	FUNCTION_BLOCK FB 324
	TITLE =G224M COUPLING DEVICE WALL GERM 7
	//COPYRIGHT:    (C) 2009  BUHLER AG, CH-9240 UZWIL, SWITZERLAND
	//
	//PRODUCT:      WinCoS_BIW01_09
	//
	//TITLE:        COUPLING DEVICE WALL GERM 7
	//                Machine group control
	//                Maschinengruppensteuerung
	//
	//--------------------------------------------------------------------------------
	//
	//IDENT:        AUTHOR:             DEPT:                              DATE:
	//
	//P01_FB324.1.0 K.Renz              CSB41                              13.Jan.2010
	//             1st Release
	//
	//--------------------------------------------------------------------------------
	//
	//PURPOSE:
	//
	//MANUAL :
	//
	//RESTRICTIONS:
	//
	//--------------------------------------------------------------------------------
	AUTHOR  : KR
	FAMILY  : USW
	VERSION : 9.9


	VAR
	  Gr       : FB10;	//Standard interface to group
	  InOutValue1    : DINT; //Data for user
	  InOutValue2    : DINT; //Data for user
	  OutWayConflict : BOOL;	//Data for user
	  OutSelectionOk : BOOL;	//Data for user
	  CmdNewValue : BOOL;	//Data for user
	  CmdNewJob   : BOOL;	//Data for user
	  OutCodeOK   : BOOL;	//Data for user
	  InEndOfJob  : BOOL ;	//Data for user
	  staWayOk      : BOOL ;	//Data for user
	  EdgeStartRelease : BOOL ;	//Data for user
	  USW8  : BOOL;	//Data for user
	  USW9 : BOOL;	//Data for user
	  USW10: BOOL;	//Data for user
	  USW11: BOOL;	//Data for user
	  USW12: BOOL;	//Data for user
	  USW13: BOOL;	//Data for user
	  USW14: BOOL;	//Data for user
	  USW15: BOOL;	//Data for user
	     #A_2715_BZS42 : FB14;   // DigInpCont
	     #A_2715_BZS43 : FB14;   // DigInpCont
	     #A_2715_BZS47 : FB14;   // DigInpCont
	     #A_2715_BZS46 : FB14;   // DigInpCont
	     #A_2715_MXZ41 : FB12;   // Motor
	     #A_2715_MXZ45 : FB12;   // Motor
	END_VAR
	VAR_TEMP
	   tmpEnable		: BOOL;
	   tmpFlag  		: BOOL;
	   tmpCmdNext		: BOOL;
	   tmpLocal  		: BOOL;
	   tmpAspOk  		: BOOL;
	   tmpHWStop 		: BOOL;
	   tmpInstanzDBNo       : INT ;
	END_VAR
	BEGIN
	NETWORK
	TITLE =
	NETWORK
	TITLE =Read command from group control
	//Parameter
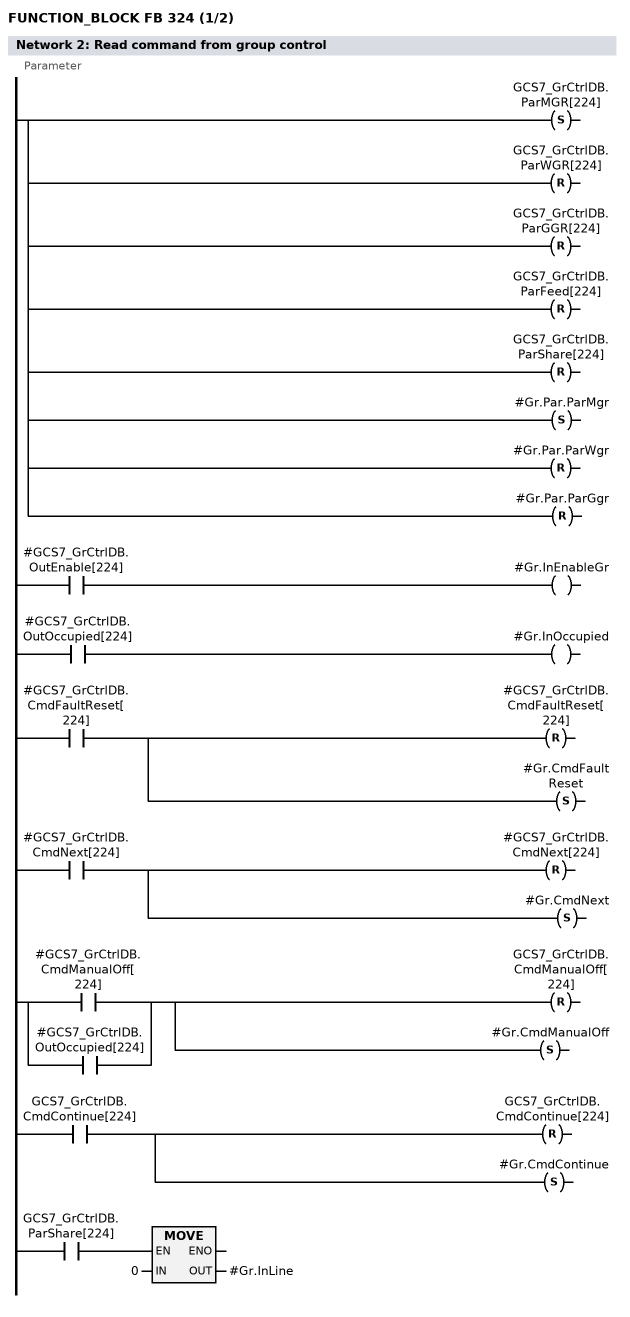
	      SET;
	      S   GCS7_GrCtrlDB.ParMGR[224];
	      R   GCS7_GrCtrlDB.ParWGR[224];
	      R   GCS7_GrCtrlDB.ParGGR[224];
	      R   GCS7_GrCtrlDB.ParFeed[224];
	      R   GCS7_GrCtrlDB.ParShare[224];
	      S   #Gr.Par.ParMgr;
	      R   #Gr.Par.ParWgr;
	      R   #Gr.Par.ParGgr;
	//Command
	      U   #GCS7_GrCtrlDB.OutEnable[224];
	      =   #Gr.InEnableGr;
	      U   #GCS7_GrCtrlDB.OutOccupied[224];
	      =   #Gr.InOccupied;
	      U   #GCS7_GrCtrlDB.CmdFaultReset[224];
	      R   #GCS7_GrCtrlDB.CmdFaultReset[224];
	      S   #Gr.CmdFaultReset;
	      U  #GCS7_GrCtrlDB.CmdNext[224];
	      R   #GCS7_GrCtrlDB.CmdNext[224];
	      S   #Gr.CmdNext;
	      U   #GCS7_GrCtrlDB.CmdManualOff[224];
	      O   #GCS7_GrCtrlDB.OutOccupied[224];
	      R   GCS7_GrCtrlDB.CmdManualOff[224];
	      S   #Gr.CmdManualOff;
	      U  GCS7_GrCtrlDB.CmdContinue[224];
	      R   GCS7_GrCtrlDB.CmdContinue[224];
	      S   #Gr.CmdContinue;
	//Init Line Number
	      U   GCS7_GrCtrlDB.ParShare[224];
	      SPBN WE00;
	      L     0;
	      T     #Gr.InLine;
	WE00: NOP   0;
	NETWORK
	TITLE =Call Methode Control
	// 1. Handle Interface PCControl
	// 2. Prepare mode --> ModePassive,ModeActive,ModeIdling
	// 3. Reset global flags of the group
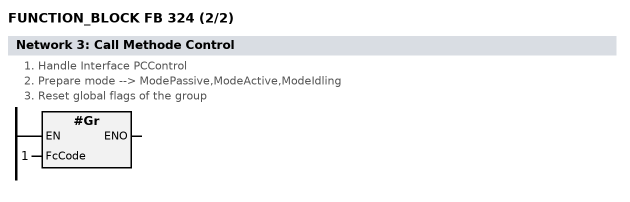
	      CALL #Gr (
	           FcCode                   := 1);
	NETWORK
	TITLE =Restart Idling Time
		L  #Gr.Par.ParIdling;
		L  2;
		>=I;
		SPB IdTm;
		T  #Gr.Par.ParIdling;
	IdTm:   NOP 0;
	      CLR;
	      S    #Gr.CmdRestartIdling;
	NETWORK
	TITLE =Prepare global flags
	NETWORK
	TITLE =Set Pattern (Target position)
	NETWORK
	TITLE =Interlocking WayOk
	//
	NETWORK
	TITLE =Interlocking Autostart
		CLR;
		R   #Gr.OutAutostart;
	NETWORK
	TITLE =Interlocking Enable
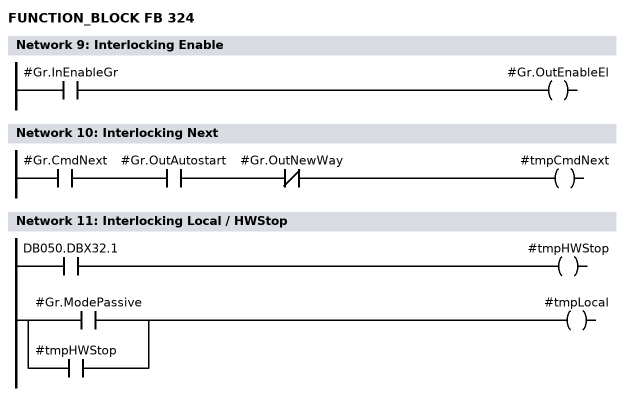
	      U     #Gr.InEnableGr;
	      =     #Gr.OutEnableEl;

	NETWORK
	TITLE =Interlocking Next
	      U     #Gr.CmdNext;
	      U     #Gr.OutAutostart;
	      UN    #Gr.OutNewWay;
	      =    #tmpCmdNext;

	NETWORK
	TITLE =Interlocking Local / HWStop
	      U    DB050.DBX32.1;
	      =    #tmpHWStop;

	      U    #Gr.ModePassive;
	      O    #tmpHWStop;
	      =    #tmpLocal;

	NETWORK
	TITLE ==A-2715-BZS42 : COUPLING DRIVE UNLOCKED
	NOP 0;
	//-InLocal---
	      U     #tmpLocal;
	      =     #A_2715_BZS42.InLocal;
	//
	//-Monitoring---
	      CLR;
	      =      #A_2715_BZS42.InMonTrue;
	      CLR;
	      =      #A_2715_BZS42.InMonFalse;
	//
	//-PreAlarm---
	      CLR;
	      =      #A_2715_BZS42.InPreAlarmTrue;
	      CLR;
	      =      #A_2715_BZS42.InPreAlarmFalse;
	//
	//-Additional commands---
	//      CLR
	//      S     #A_2715_BZS42.CmdRunTimeOutTime
	//
	//-Read inputs---
	      U     E 763.0;
	      =     #A_2715_BZS42.InpTrue;
	      U   DB050.DBX32.1;
	      =     #A_2715_BZS42.InHWStop;
	       U     PLC_DPInfo.Master[1].SlavesError[75];
	       =       #A_2715_BZS42.InDPFault;
	//
	//-Set Parameters---
	//
	//-Call object control---
	      CALL  #A_2715_BZS42;
	//
	//-Write outputs---
	NETWORK
	TITLE ==A-2715-BZS43 : COUPLING DRIVE LOCKED
	NOP 0;
	//-InLocal---
	      U     #tmpLocal;
	      =     #A_2715_BZS43.InLocal;
	//
	//-Monitoring---
	      CLR;
	      =      #A_2715_BZS43.InMonTrue;
	      CLR;
	      =      #A_2715_BZS43.InMonFalse;
	//
	//-PreAlarm---
	      CLR;
	      =      #A_2715_BZS43.InPreAlarmTrue;
	      CLR;
	      =      #A_2715_BZS43.InPreAlarmFalse;
	//
	//-Additional commands---
	//      CLR
	//      S     #A_2715_BZS43.CmdRunTimeOutTime
	//
	//-Read inputs---
	      U     E 763.1;
	      =     #A_2715_BZS43.InpTrue;
	      U   DB050.DBX32.1;
	      =     #A_2715_BZS43.InHWStop;
	       U     PLC_DPInfo.Master[1].SlavesError[75];
	       =       #A_2715_BZS43.InDPFault;
	//
	//-Set Parameters---
	//
	//-Call object control---
	      CALL  #A_2715_BZS43;
	//
	//-Write outputs---
	NETWORK
	TITLE ==A-2715-BZS47 : COUPLING DRIVE LOCKED
	NOP 0;
	//-InLocal---
	      U     #tmpLocal;
	      =     #A_2715_BZS47.InLocal;
	//
	//-Monitoring---
	      CLR;
	      =      #A_2715_BZS47.InMonTrue;
	      CLR;
	      =      #A_2715_BZS47.InMonFalse;
	//
	//-PreAlarm---
	      CLR;
	      =      #A_2715_BZS47.InPreAlarmTrue;
	      CLR;
	      =      #A_2715_BZS47.InPreAlarmFalse;
	//
	//-Additional commands---
	//      CLR
	//      S     #A_2715_BZS47.CmdRunTimeOutTime
	//
	//-Read inputs---
	      U     E 763.3;
	      =     #A_2715_BZS47.InpTrue;
	      U   DB050.DBX32.1;
	      =     #A_2715_BZS47.InHWStop;
	       U     PLC_DPInfo.Master[1].SlavesError[75];
	       =       #A_2715_BZS47.InDPFault;
	//
	//-Set Parameters---
	//
	//-Call object control---
	      CALL  #A_2715_BZS47;
	//
	//-Write outputs---
	NETWORK
	TITLE ==A-2715-BZS46 : COUPLING DRIVE UNLOCKED
	NOP 0;
	//-InLocal---
	      U     #tmpLocal;
	      =     #A_2715_BZS46.InLocal;
	//
	//-Monitoring---
	      CLR;
	      =      #A_2715_BZS46.InMonTrue;
	      CLR;
	      =      #A_2715_BZS46.InMonFalse;
	//
	//-PreAlarm---
	      CLR;
	      =      #A_2715_BZS46.InPreAlarmTrue;
	      CLR;
	      =      #A_2715_BZS46.InPreAlarmFalse;
	//
	//-Additional commands---
	//      CLR
	//      S     #A_2715_BZS46.CmdRunTimeOutTime
	//
	//-Read inputs---
	      U     E 763.2;
	      =     #A_2715_BZS46.InpTrue;
	      U   DB050.DBX32.1;
	      =     #A_2715_BZS46.InHWStop;
	       U     PLC_DPInfo.Master[1].SlavesError[75];
	       =       #A_2715_BZS46.InDPFault;
	//
	//-Set Parameters---
	//
	//-Call object control---
	      CALL  #A_2715_BZS46;
	//
	//-Write outputs---
	NETWORK
	TITLE ==A-2715-MXZ41 : WALL COUPLING DRIVE
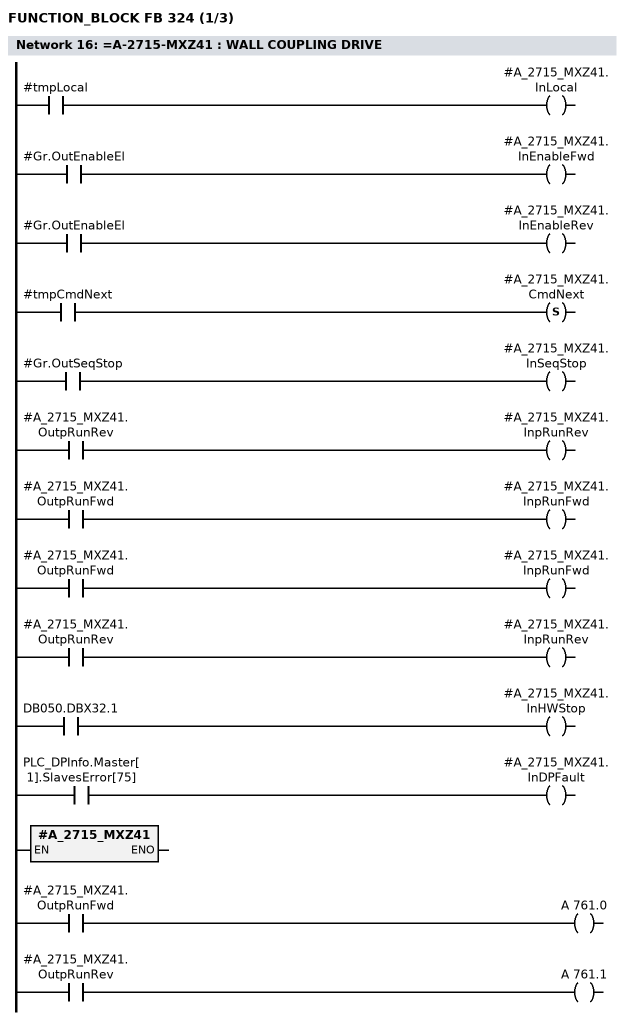
	NOP 0;
	//-InLocal---
	      U     #tmpLocal;
	      =     #A_2715_MXZ41.InLocal;
	//
	//-Interlocking---
	      U     #Gr.OutEnableEl;
	      =     #A_2715_MXZ41.InEnableFwd;
	      U     #Gr.OutEnableEl;
	      =     #A_2715_MXZ41.InEnableRev;
	//
	      U    #tmpCmdNext;
	      S     #A_2715_MXZ41.CmdNext;
	//
	      U     #Gr.OutSeqStop;
	      =     #A_2715_MXZ41.InSeqStop;
	//
	//-Read inputs---
	      U     #A_2715_MXZ41.OutpRunRev;
	      =     #A_2715_MXZ41.InpRunRev;
	      U     #A_2715_MXZ41.OutpRunFwd;
	      =     #A_2715_MXZ41.InpRunFwd;
	      U     #A_2715_MXZ41.OutpRunFwd;
	      =     #A_2715_MXZ41.InpRunFwd;
	      U     #A_2715_MXZ41.OutpRunRev;
	      =     #A_2715_MXZ41.InpRunRev;
	      U   DB050.DBX32.1;
	      =     #A_2715_MXZ41.InHWStop;
	       U     PLC_DPInfo.Master[1].SlavesError[75];
	       =       #A_2715_MXZ41.InDPFault;
	//
	//-Set Parameters---
	//
	//-Call object control---
	      CALL  #A_2715_MXZ41;
	//
	//-Write outputs---
	      U     #A_2715_MXZ41.OutpRunFwd;
	      =     A 761.0;
	      U     #A_2715_MXZ41.OutpRunRev;
	      =     A 761.1;
	NETWORK
	TITLE ==A-2715-MXZ45 : WALL COUPLING DRIVE
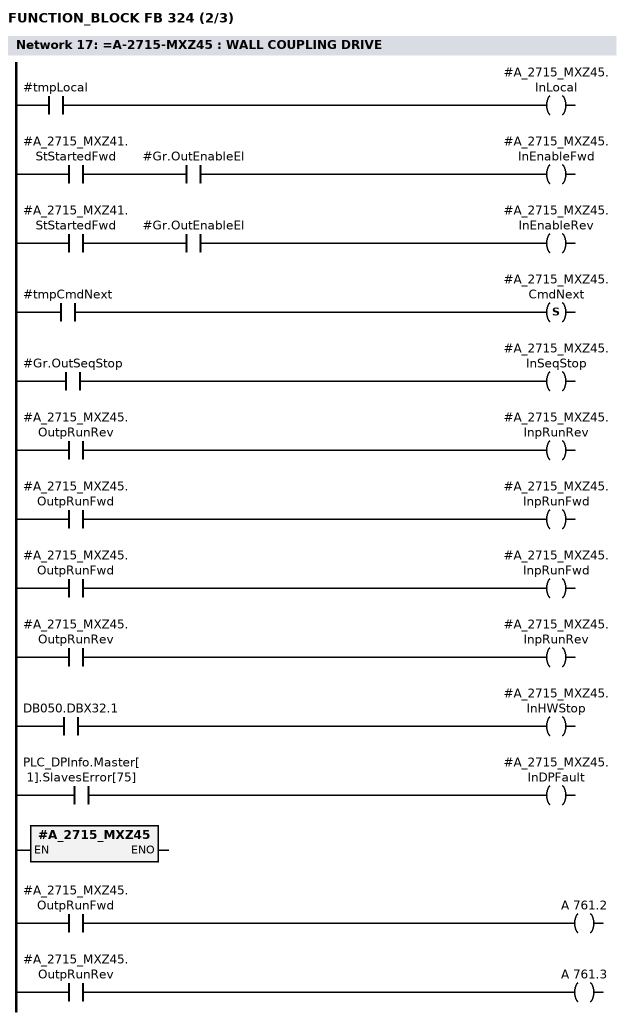
	NOP 0;
	//-InLocal---
	      U     #tmpLocal;
	      =     #A_2715_MXZ45.InLocal;
	//
	//-Interlocking---
	      U     #A_2715_MXZ41.StStartedFwd;
	      U     #Gr.OutEnableEl;
	      =     #A_2715_MXZ45.InEnableFwd;
	      U     #A_2715_MXZ41.StStartedFwd;
	      U     #Gr.OutEnableEl;
	      =     #A_2715_MXZ45.InEnableRev;
	//
	      U    #tmpCmdNext;
	      S     #A_2715_MXZ45.CmdNext;
	//
	      U     #Gr.OutSeqStop;
	      =     #A_2715_MXZ45.InSeqStop;
	//
	//-Read inputs---
	      U     #A_2715_MXZ45.OutpRunRev;
	      =     #A_2715_MXZ45.InpRunRev;
	      U     #A_2715_MXZ45.OutpRunFwd;
	      =     #A_2715_MXZ45.InpRunFwd;
	      U     #A_2715_MXZ45.OutpRunFwd;
	      =     #A_2715_MXZ45.InpRunFwd;
	      U     #A_2715_MXZ45.OutpRunRev;
	      =     #A_2715_MXZ45.InpRunRev;
	      U   DB050.DBX32.1;
	      =     #A_2715_MXZ45.InHWStop;
	       U     PLC_DPInfo.Master[1].SlavesError[75];
	       =       #A_2715_MXZ45.InDPFault;
	//
	//-Set Parameters---
	//
	//-Call object control---
	      CALL  #A_2715_MXZ45;
	//
	//-Write outputs---
	      U     #A_2715_MXZ45.OutpRunFwd;
	      =     A 761.2;
	      U     #A_2715_MXZ45.OutpRunRev;
	      =     A 761.3;
	NETWORK
	TITLE =Test Fault
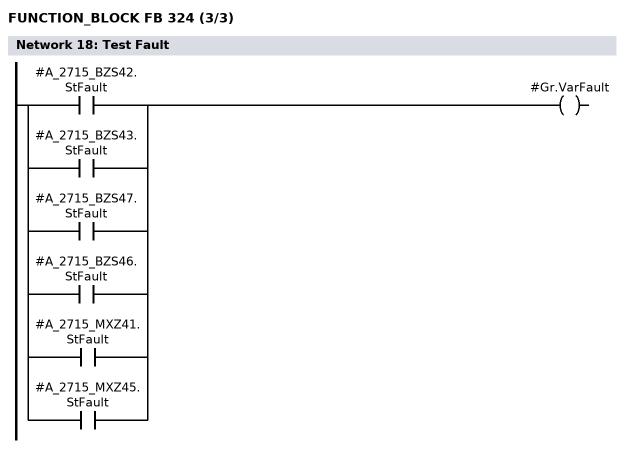
	      U     #A_2715_BZS42.StFault;
	      O     #A_2715_BZS43.StFault;
	      O     #A_2715_BZS47.StFault;
	      O     #A_2715_BZS46.StFault;
	      O     #A_2715_MXZ41.StFault;
	      O     #A_2715_MXZ45.StFault;
	      =     #Gr.VarFault;
	NETWORK
	TITLE =Test Warning
	      CLR;
	      =     #Gr.OutWarning;
	NETWORK
	TITLE =Test Stopped
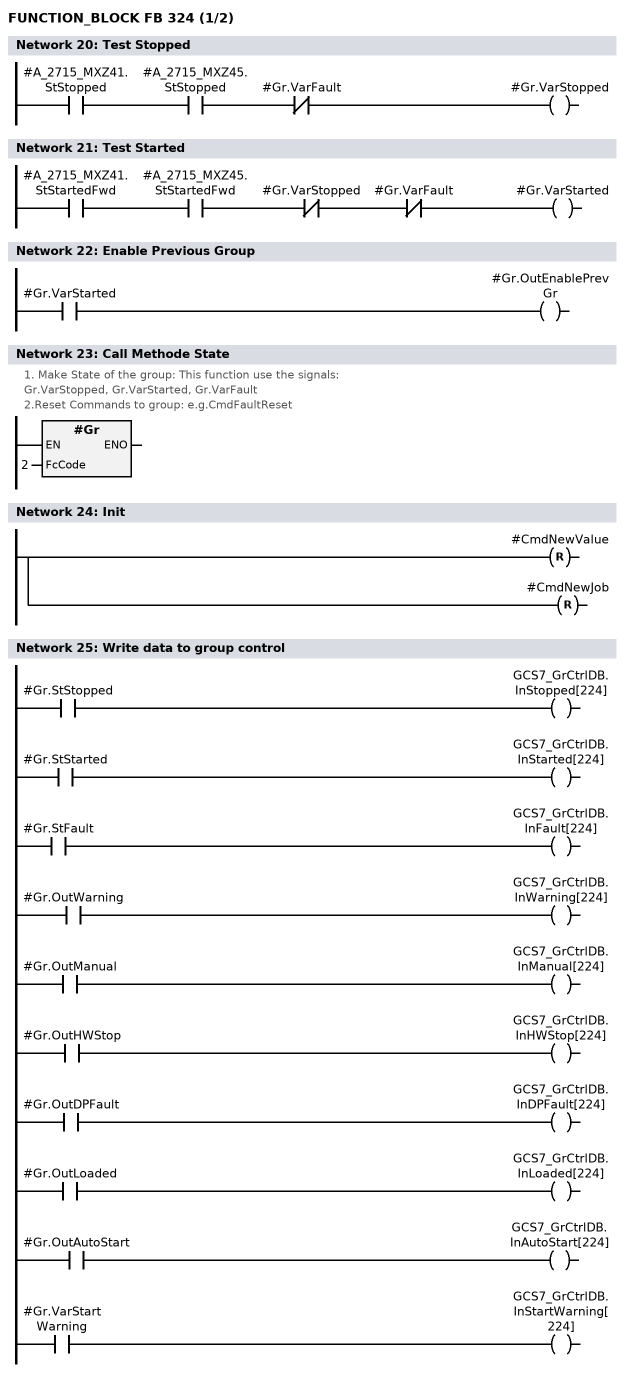
	      U     #A_2715_MXZ41.StStopped;
	      U     #A_2715_MXZ45.StStopped;
	      UN   #Gr.VarFault;
	      =     #Gr.VarStopped;
	NETWORK
	TITLE =Test Started
	      U     #A_2715_MXZ41.StStartedFwd;
	      U     #A_2715_MXZ45.StStartedFwd;
	      UN  #Gr.VarStopped;
	      UN  #Gr.VarFault;
	      =     #Gr.VarStarted;
	NETWORK
	TITLE =Enable Previous Group
	      U    #Gr.VarStarted;
	      =     #Gr.OutEnablePrevGr;
	NETWORK
	TITLE =Call Methode State
	//1. Make State of the group: This function use the signals:
	//        Gr.VarStopped, Gr.VarStarted, Gr.VarFault
	//2.Reset Commands to group: e.g.CmdFaultReset
	      CALL #Gr (
	           FcCode                   := 2);
	NETWORK
	TITLE =Init
	      SET;
	      R    #CmdNewValue;
	      R    #CmdNewJob;
	NETWORK
	TITLE =Write data to group control
	      U   #Gr.StStopped;
	      =   GCS7_GrCtrlDB.InStopped[224];
	      U   #Gr.StStarted;
	      =   GCS7_GrCtrlDB.InStarted[224];
	      U   #Gr.StFault;
	      =   GCS7_GrCtrlDB.InFault[224];
	      U   #Gr.OutWarning;
	      =   GCS7_GrCtrlDB.InWarning[224];
	      U   #Gr.OutManual;
	      =   GCS7_GrCtrlDB.InManual[224];
	      U   #Gr.OutHWStop;
	      =   GCS7_GrCtrlDB.InHWStop[224];
	      U   #Gr.OutDPFault;
	      =   GCS7_GrCtrlDB.InDPFault[224];
	      U   #Gr.OutLoaded;
	      =   GCS7_GrCtrlDB.InLoaded[224];
	      U   #Gr.OutAutoStart;
	      =   GCS7_GrCtrlDB.InAutoStart[224];
	      U   #Gr.VarStartWarning;
	      =   GCS7_GrCtrlDB.InStartWarning[224];
	NETWORK
	TITLE =End of block
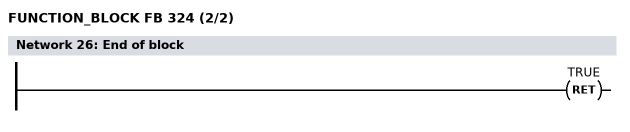

	BE

	END_FUNCTION_BLOCK
